(* IEC 61131-3 sources: Caravan/Stations/Terminal/HMI/Class/Koordinates_Class, 1 file *)

(* ---- Koordinates_Class.st ---- *)
(*!
<Class
	Name               = "Koordinates_Class"
	Revision           = "0.0"
	RealtimeTask       = "false"
	CyclicTask         = "true"
	DefCyclictime      = "100 ms"
	BackgroundTask     = "false"
	Sigmatek           = "false"
	OSInterface        = "false"
	HighPriority       = "false"
	Automatic          = "false"
	UpdateMode         = "Prescan"
	SharedCommandTable = "true"
	Objectsize         = "(660,240)">
	<Channels>
		<Server Name="ClassSvr" Visualized="false" Initialize="false" WriteProtected="true" Retentive="false"/>
		<Client Name="Input_X_C" Required="true" Internal="false"/>
		<Client Name="Input_Y_C" Required="true" Internal="false"/>
		<Client Name="Output_X_C" Required="true" Internal="false"/>
		<Client Name="Output_Y_C" Required="true" Internal="false"/>
	</Channels>
</Class>
*)
Koordinates_Class : CLASS
  //Servers:
	ClassSvr 	: SvrChCmd_DINT;
  //Clients:
	Input_X_C 	: CltCh_DINT;
	Input_Y_C 	: CltCh_DINT;
	Output_X_C 	: CltCh_DINT;
	Output_Y_C 	: CltCh_DINT;
  //Variables:
  //Functions:

	FUNCTION VIRTUAL GLOBAL CyWork
		VAR_INPUT
			EAX 	: UDINT;
		END_VAR
		VAR_OUTPUT
			state (EAX) 	: UDINT;
		END_VAR;
  //Tables:
	FUNCTION @STD
		VAR_OUTPUT
			ret_code	: CONFSTATES;
		END_VAR;
	FUNCTION GLOBAL TAB @CT_;
END_CLASS;

FUNCTION VIRTUAL GLOBAL Koordinates_Class::CyWork
	VAR_INPUT
		EAX 	: UDINT;
	END_VAR
	VAR_OUTPUT
		state (EAX) 	: UDINT;
	END_VAR

      Input_X_C   :=    Input_X_C.Read();
      Input_Y_C   :=    Input_Y_C.Read();

      Output_X_C    :=    Output_X_C.Write(input:=Input_X_C);
      Output_Y_C    :=    Output_Y_C.Write(input:=Input_Y_C);

	state := READY;

END_FUNCTION
